// TIA Portal V20 export
// export: Created 2026-07-10T11:12:29.5776723Z, ExportSetting WithDefaults, DisplayName Totally Integrated Automation Portal, DisplayVersion V20, DisplayName TIA Portal Openness, DisplayVersion V20, DisplayName TIA Portal Version Control Interface, DisplayVersion V20, DisplayName STEP 7 Professional, DisplayVersion V20, DisplayName STEP 7 Safety, DisplayVersion V20, DisplayName WinCC Basic/Comfort/Advanced, DisplayVersion V20, DisplayName WinCC Unified, DisplayVersion V20
DATA_BLOCK "ModbusClO2_DB"   // DB7
VERSION : 0.1
// stored: AutoNumber true, DBAccessibleFromOPCUA true, InstanceOfName ModbusClO2, InstanceOfType FB
"ModbusClO2"
   // VAR
   //    ProportionalDosingExternal { S7_SetPoint := 'True'} : DWord;
   //    AbsoluteDosing : DWord;
   //    SystemProductivity : DWord;
   //    Pressure : Word;
   //    Doser1Productivity : Word;
   //    Doser2Productivity : Word;
   // END_VAR
BEGIN
END_DATA_BLOCK
